// TIA Portal V17 export
// export: Created 2022-04-06T07:28:41.5576845Z, ExportSetting WithDefaults, DisplayName Totally Integrated Automation Portal, DisplayVersion V17, DisplayName TIA Portal Openness, DisplayVersion V17, DisplayName TIA Portal Version Control Interface, DisplayVersion V17, DisplayName TIA Portal Test Suite Advanced, DisplayVersion V17, DisplayName SINAMICS Startdrive Advanced, DisplayVersion V17, DisplayName SINAMICS Startdrive G130, G150, S120, S150, SINAMICS MV, S210, DisplayVersion V17, DisplayName SINAMICS Startdrive G110M, G120, G120C, G120D, G120P, G115D, DisplayVersion V17, DisplayName STEP 7 Professional, DisplayVersion V17, DisplayName STEP 7 Safety, DisplayVersion V17, DisplayName WinCC Advanced / Unified PC, DisplayVersion V17
TYPE "LAxisCtrl_typePosSuperimposed"
TITLE = LAxisCtrl_typePosSuperimposed
// Support: tech.team.motioncontrol@siemens.com
// stored: IsFailsafeCompliant false
   STRUCT
      distance : LReal := 0.0;   // Distance for superimposed positioning
      velocityDiff : LReal := -1.0;   // Maximum velocity deviation compared to the active motion (Value > 0.0: The specified value is used; Value = 0.0: Not permitted; Value < 0.0: Use of the default value configured in the technology object)
      acceleration : LReal := -1.0;   // Acceleration for positioning (Value > 0.0: The specified value is used; Value = 0.0: Not permitted; Value < 0.0: Use of the default value configured in the technology object)
      deceleration : LReal := -1.0;   // Deceleration for positioning (Value > 0.0: The specified value is used; Value = 0.0: Not permitted; Value < 0.0: Use of the default value configured in the technology object)
      jerk : LReal := -1.0;   // Jerk for positioning (Value > 0.0: Smooth velocity profile, the specified value is used; Value = 0.0: Trapezoid velocity profile; Value < 0.0: Use of the default value configured in the technology object)
      direction : DInt := 0;   // Motion direction of the axis (0: The sign of the distance parameter defines the direction; 1: Positive negative; 2: Negative direction)
   END_STRUCT;
END_TYPE
